{attribute 'linkalways'} 
{attribute 'no_explicit_call' := 'This FB is a CLASS and must be accessed using methods or properties'}
{attribute 'enable_dynamic_creation'}
FUNCTION_BLOCK _ETcVnStructuringElementShape EXTENDS EnumDatatypeBase
VAR
	localData : ETcVnStructuringElementShape;
	activeData : REFERENCE TO ETcVnStructuringElementShape;
	enumBaseDatatype : _DINT(localData);
END_VAR

METHOD PRIVATE AddLocalEnumeration
VAR_INPUT
	Enumeration : T_MAXSTRING;
	Value : ETcVnStructuringElementShape;
END_VAR
AddEnumeration(Enumeration, Value);
END_METHOD

PROPERTY PUBLIC Address : PVOID
GET
Address := ADR(activeData);
END_GET
END_PROPERTY

METHOD PUBLIC ClearReference
VAR_INPUT
END_VAR
activeData REF= localData;
SetBaseDatatypeReference();
END_METHOD

METHOD PUBLIC Clone : I_Datatype
VAR
    pClone : POINTER TO _ETcVnStructuringElementShape;
END_VAR
pClone := __NEW(_ETcVnStructuringElementShape(InitialValue := Value));
Clone := pClone^;
END_METHOD

METHOD FB_init : BOOL
VAR_INPUT
	bInitRetains : BOOL; // if TRUE, the retain variables are initialized (warm start / cold start)
	bInCopyCode : BOOL;  // if TRUE, the instance afterwards gets moved into the copy code (online change)
	InitialValue : ETcVnStructuringElementShape;
END_VAR
localData := InitialValue;
AddBaseDatatype(enumBaseDatatype);
ClearReference();

AddLocalEnumeration('TCVN_SES_RECTANGLE', ETcVnStructuringElementShape.TCVN_SES_RECTANGLE);
AddLocalEnumeration('TCVN_SES_CROSS', ETcVnStructuringElementShape.TCVN_SES_CROSS);
AddLocalEnumeration('TCVN_SES_ELLIPSE', ETcVnStructuringElementShape.TCVN_SES_ELLIPSE);
END_METHOD

PROPERTY PUBLIC Identifier : T_MAXSTRING
GET
Identifier := 'ETcVnStructuringElementShape';
END_GET
END_PROPERTY

METHOD IsEnumeratorValueEqual : BOOL
VAR_INPUT
	Enumerator : I_KeyValueForwardEnumerator;
END_VAR
VAR
	storedValue : ETcVnStructuringElementShape;
END_VAR
IF NOT Enumerator.TryGet(storedValue) THEN
	RETURN;
END_IF

IsEnumeratorValueEqual := storedValue = activeData;
END_METHOD

METHOD PUBLIC MakeReferenceTo
VAR_INPUT
	ReferenceTarget : REFERENCE TO ETcVnStructuringElementShape;
END_VAR
activeData REF= ReferenceTarget;
SetBaseDatatypeReference();
END_METHOD

METHOD PROTECTED SetBaseDatatypeReference
VAR_INPUT
END_VAR
enumBaseDatatype.MakeReferenceTo(activeData);
END_METHOD

PROPERTY PUBLIC Size : UDINT
GET
Size := SIZEOF(activeData);
END_GET
END_PROPERTY

METHOD TryMakeReferenceTo : BOOL
VAR_INPUT
	Target : I_Datatype;
END_VAR
VAR
	targetAsEnum : I_EnumDatatype;
	pTargetData : POINTER TO ETcVnStructuringElementShape;
END_VAR
IF NOT Target.TryResolveAsEnumDatatype(targetAsEnum) THEN
	RETURN;
END_IF

IF targetAsEnum.Identifier <> Identifier THEN
	RETURN;
END_IF

pTargetData := Target.Address;
activeData REF= pTargetData^;
SetBaseDatatypeReference();
TryMakeReferenceTo := TRUE;
END_METHOD

PROPERTY PUBLIC Value : ETcVnStructuringElementShape
GET
Value := activeData;
END_GET
SET
activeData := Value;
END_SET
END_PROPERTY

END_FUNCTION_BLOCK

(* stored: Version 1.1.0.1, ProductVersion 3.1.4024.12
   POU _ETcVnStructuringElementShape: Id {98728f69-0608-0d2b-10b0-74611e94f838}, SpecialFunc None
   Folder Constructor: Id {b1c8afc6-282a-0502-215b-d81ce3079bd8}
   Folder Private: Id {cb20952e-2cdf-0515-2b56-db8d43aa7dea}
   Folder Protected: Id {d4b3f6cc-e452-0aad-1187-e9dabdee7998}
   Method AddLocalEnumeration: Id {5c0beae6-790d-0715-1fbc-e987da497e9f}
   Property Address: Id {68e66a30-8fcb-0380-33dd-e4d185e1c6c4}
   Get Get: Id {70d046f9-4ba7-09fc-0782-5ee8badaec9c}
   Method ClearReference: Id {eab77c0c-96d5-0bc4-3400-b429c21375e8}
   Method Clone: Id {7f29dc26-3af6-0c8d-06c1-be66f7382347}
   Method FB_init: Id {26b61613-c7e1-0a0b-0ea4-aab97e68ca7b}
   Property Identifier: Id {1c4a4fd8-d362-02f8-3be8-c8bdf926fddb}
   Get Get: Id {71467f8e-8dd6-0ce5-3345-12339c5cbe75}
   Method IsEnumeratorValueEqual: Id {a3a3020d-5216-044e-15ca-119adee6a51d}
   Method MakeReferenceTo: Id {52082723-81d8-07b5-27fd-305501175631}
   Method SetBaseDatatypeReference: Id {4daf3b95-b0b2-07f4-2432-a4286c07d7f7}
   Property Size: Id {8f445e42-2ed1-0a73-324f-2415cfacff09}
   Get Get: Id {7e1c981e-8bce-069c-3b1b-786e3a019b92}
   Method TryMakeReferenceTo: Id {722d836a-9c9a-087b-0562-d8772856cecb}
   Property Value: Id {812f6903-e6a4-0b4f-17a3-d7683961751f}
   Get Get: Id {7bcfe54d-991d-0b1b-0158-c526ef4f0857}
   Set Set: Id {511a79fe-34cc-0abb-1a51-057fd8b724bd} *)
